# EPICS autosave request: iocBoot/ioc13idd_linux/auto_positions.req
file "CARS_motor_positions.req",         P=$(P), M=m81
file "CARS_motor_positions.req",         P=$(P), M=m83
file "CARS_motor_positions.req",         P=$(P), M=m82
file "CARS_motor_positions.req",         P=$(P), M=m84
file "CARS_motor_positions.req",         P=$(P), M=m94
file "CARS_motor_positions.req",         P=$(P), M=m93
